// TIA Portal V17 export
// export: Created 2025-03-13T10:30:20.791718Z, ExportSetting WithDefaults, DisplayName Totally Integrated Automation Portal, DisplayVersion V17 Update 8, DisplayName TIA Portal Openness, DisplayVersion V17 Update 8, DisplayName TIA Portal Version Control Interface, DisplayVersion V17, DisplayName SINAMICS Startdrive Advanced, DisplayVersion V17 SP2, DisplayName SINAMICS Startdrive G110M, G120, G120C, G120D, G120P, G115D, DisplayVersion V17 SP2, DisplayName SINAMICS Startdrive G130, G150, S120, S150, SINAMICS MV, S210, DisplayVersion V17 SP2, DisplayName STEP 7 Professional, DisplayVersion V17 Update 8, DisplayName SINUMERIK ONE STEP 7 Toolbox, DisplayVersion V17 Update 12, DisplayName SINUMERIK 840D sl STEP 7 Toolbox, DisplayVersion V17 Update 12, DisplayName STEP 7 Safety, DisplayVersion V17 Update 6, DisplayName WinCC Advanced, DisplayVersion V17 Update 8
FUNCTION "UPTL_DirectKeys" : Void   // FC1057, LAD
{ S7_Optimized_Access := 'FALSE' }
AUTHOR : Transline
FAMILY : UPTL_Transline
VERSION : 4.0
// stored: AutoNumber true, IsIECCheckEnabled false, SetENOAutomatically false, UDAEnableTagReadback false
   VAR_TEMP
      tmpCollect : Bool;
      tmpPlusKeys : Byte;
      tmpMinusKeys : Byte;
      tmpRetVal : Word;
   END_VAR
BEGIN

REGION Network 1: MPP-ITC-HT10 PLUS-MINUS SOFTKEYS ADDRESSES
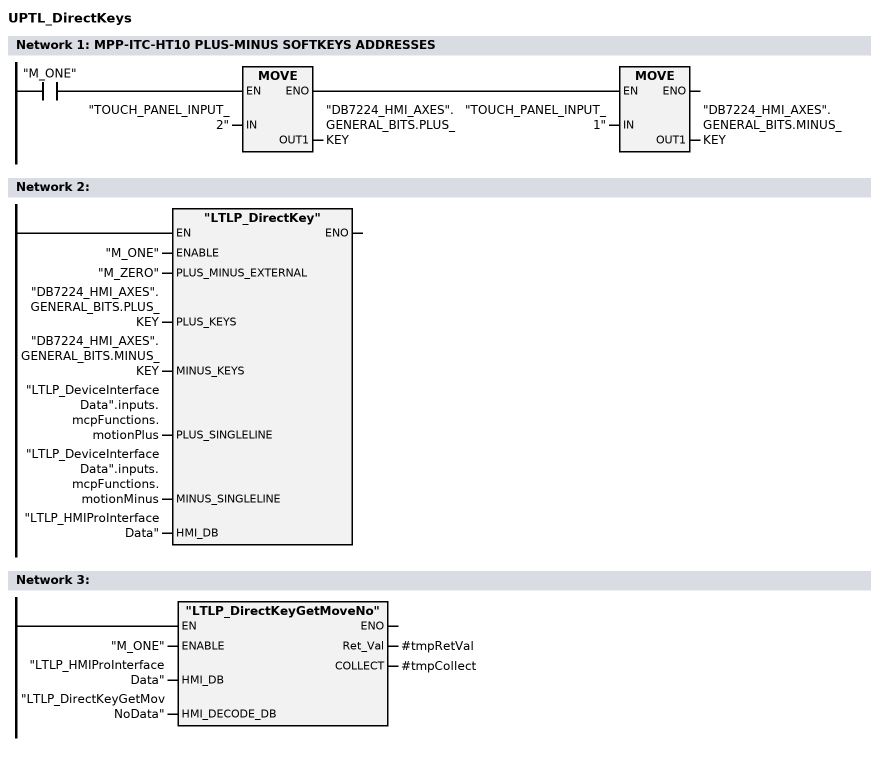
   RUNG wire#powerrail
      Contact( "M_ONE" )
      { S7_GenerateENO := "TRUE" } Move(in := "TOUCH_PANEL_INPUT_2", out1 => "DB7224_HMI_AXES".GENERAL_BITS.PLUS_KEY)
      { S7_GenerateENO := "TRUE" } Move(in := "TOUCH_PANEL_INPUT_1", out1 => "DB7224_HMI_AXES".GENERAL_BITS.MINUS_KEY)
   END_RUNG
   // the same network as SCL:
   // ENO of a box is taken as its EN; it also drops when the box reports an error
   IF "M_ONE" THEN
       "DB7224_HMI_AXES".GENERAL_BITS.PLUS_KEY := "TOUCH_PANEL_INPUT_2";
       "DB7224_HMI_AXES".GENERAL_BITS.MINUS_KEY := "TOUCH_PANEL_INPUT_1";
   END_IF;
END_REGION

REGION Network 2
   RUNG wire#powerrail
      "LTLP_DirectKey"(ENABLE := "M_ONE", PLUS_MINUS_EXTERNAL := "M_ZERO", PLUS_KEYS := "DB7224_HMI_AXES".GENERAL_BITS.PLUS_KEY, MINUS_KEYS := "DB7224_HMI_AXES".GENERAL_BITS.MINUS_KEY, PLUS_SINGLELINE := "LTLP_DeviceInterfaceData".inputs.mcpFunctions.motionPlus, MINUS_SINGLELINE := "LTLP_DeviceInterfaceData".inputs.mcpFunctions.motionMinus, HMI_DB := "LTLP_HMIProInterfaceData")
   END_RUNG
   // the same network as SCL:
   "LTLP_DirectKey"(ENABLE := "M_ONE",
                    PLUS_MINUS_EXTERNAL := "M_ZERO",
                    PLUS_KEYS := "DB7224_HMI_AXES".GENERAL_BITS.PLUS_KEY,
                    MINUS_KEYS := "DB7224_HMI_AXES".GENERAL_BITS.MINUS_KEY,
                    PLUS_SINGLELINE := "LTLP_DeviceInterfaceData".inputs.mcpFunctions.motionPlus,
                    MINUS_SINGLELINE := "LTLP_DeviceInterfaceData".inputs.mcpFunctions.motionMinus,
                    HMI_DB := "LTLP_HMIProInterfaceData");
END_REGION

REGION Network 3
   RUNG wire#powerrail
      "LTLP_DirectKeyGetMoveNo"(ENABLE := "M_ONE", HMI_DB := "LTLP_HMIProInterfaceData", HMI_DECODE_DB := "LTLP_DirectKeyGetMovNoData", Ret_Val => #tmpRetVal, COLLECT => #tmpCollect)
   END_RUNG
   // the same network as SCL:
   #tmpRetVal := "LTLP_DirectKeyGetMoveNo"(ENABLE := "M_ONE",
                           HMI_DB := "LTLP_HMIProInterfaceData",
                           HMI_DECODE_DB := "LTLP_DirectKeyGetMovNoData",
                           COLLECT => #tmpCollect);
END_REGION
END_FUNCTION
